// SIMATIC S7-200 SMART project (STEP 7-Micro/WIN SMART), CPU ST40

SYMBOL_TABLE 系统符号
Clock_1s         SM0.5    // 针对 1 s 的周期时间，时钟脉冲接通 0.5 s，断开 0.5 s.
END_SYMBOL_TABLE

ORGANIZATION_BLOCK MAIN:OB1
TITLE=程序注释
BEGIN
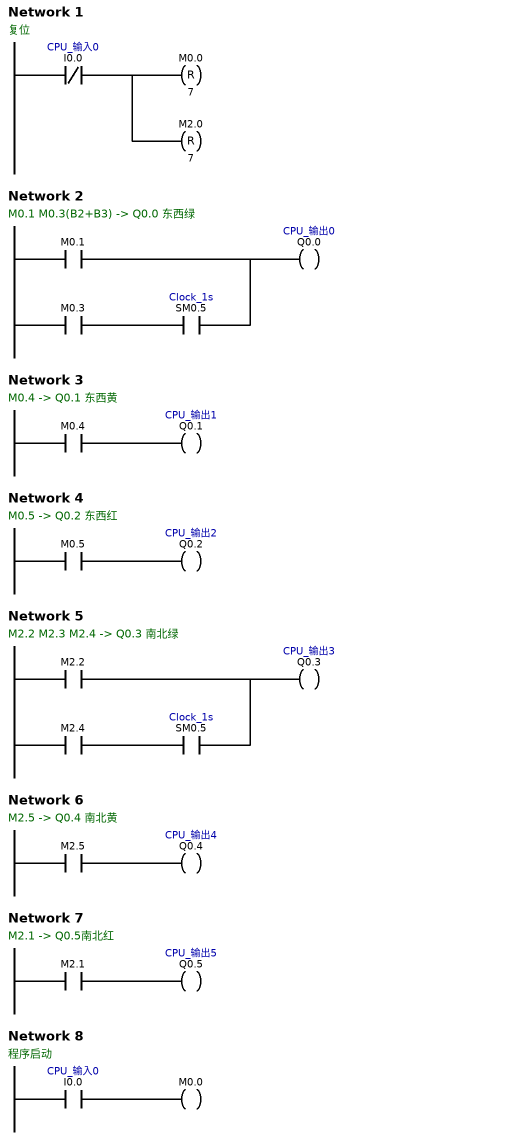
Network 1
// 复位
LDN    CPU_输入0:I0.0
R      M0.0, 7
R      M2.0, 7
Network 2
// M0.1 M0.3(B2+B3) -> Q0.0 东西绿
LD     M0.1
LD     M0.3
A      Clock_1s:SM0.5
OLD
=      CPU_输出0:Q0.0
Network 3
// M0.4 -> Q0.1 东西黄
LD     M0.4
=      CPU_输出1:Q0.1
Network 4
// M0.5 -> Q0.2 东西红
LD     M0.5
=      CPU_输出2:Q0.2
Network 5
// M2.2 M2.3 M2.4 -> Q0.3 南北绿
LD     M2.2
LD     M2.4
A      Clock_1s:SM0.5
OLD
=      CPU_输出3:Q0.3
Network 6
// M2.5 -> Q0.4 南北黄
LD     M2.5
=      CPU_输出4:Q0.4
Network 7
// M2.1 -> Q0.5南北红
LD     M2.1
=      CPU_输出5:Q0.5
Network 8
// 程序启动
LD     CPU_输入0:I0.0
=      M0.0
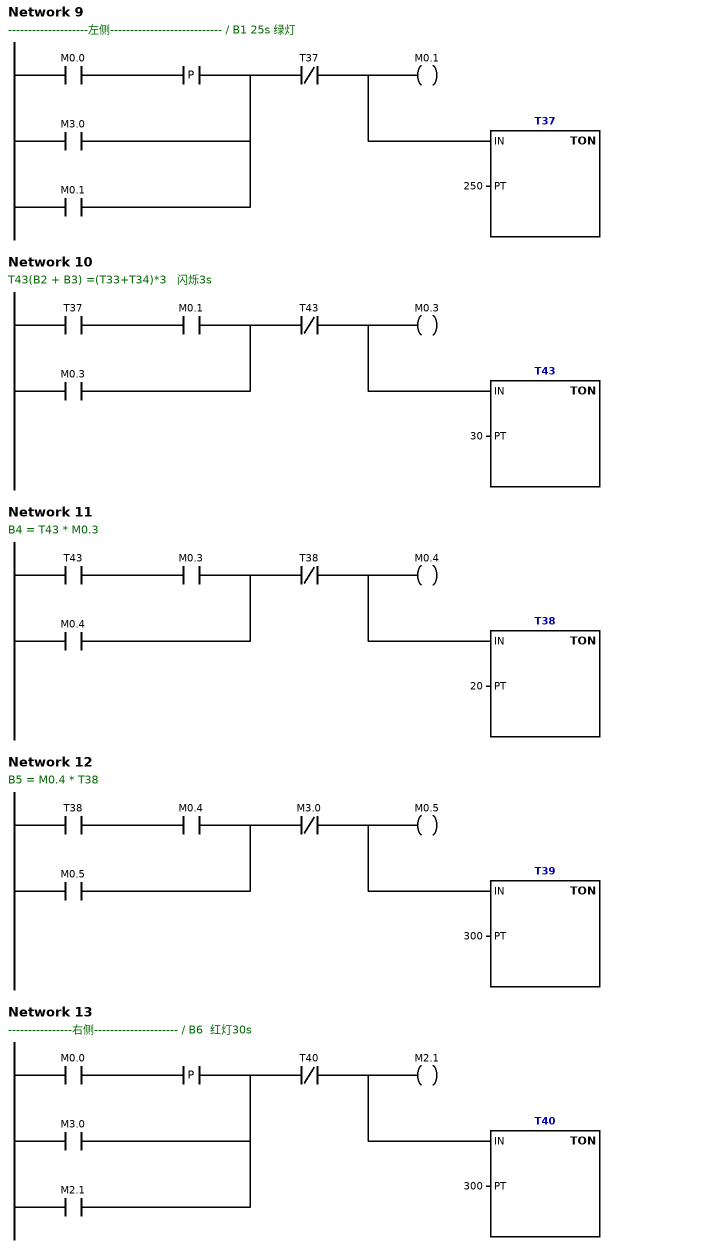
Network 9
// --------------------左侧----------------------------
// B1 25s 绿灯 
LD     M0.0
EU
O      M3.0
O      M0.1
AN     T37
=      M0.1
TON    T37, 250
Network 10
// T43(B2 + B3) =(T33+T34)*3   闪烁3s
LD     T37
A      M0.1
O      M0.3
AN     T43
=      M0.3
TON    T43, 30
Network 11
// B4 = T43 * M0.3
LD     T43
A      M0.3
O      M0.4
AN     T38
=      M0.4
TON    T38, 20
Network 12
// B5 = M0.4 * T38 
LD     T38
A      M0.4
O      M0.5
AN     M3.0
=      M0.5
TON    T39, 300
Network 13
// ----------------右侧---------------------
// B6  红灯30s
LD     M0.0
EU
O      M3.0
O      M2.1
AN     T40
=      M2.1
TON    T40, 300
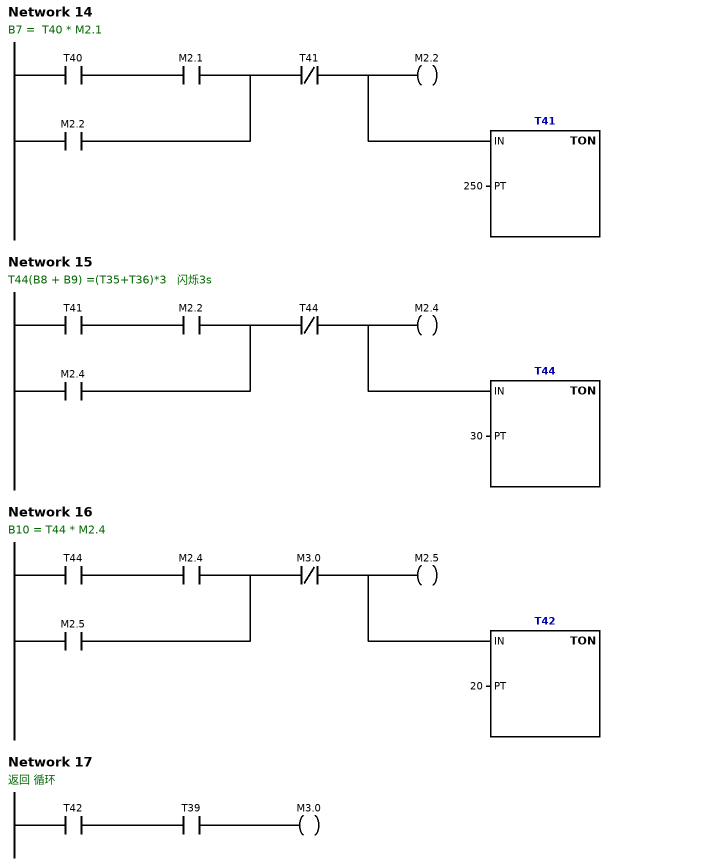
Network 14
// B7 =  T40 * M2.1
LD     T40
A      M2.1
O      M2.2
AN     T41
=      M2.2
TON    T41, 250
Network 15
// T44(B8 + B9) =(T35+T36)*3   闪烁3s
LD     T41
A      M2.2
O      M2.4
AN     T44
=      M2.4
TON    T44, 30
Network 16
// B10 = T44 * M2.4
LD     T44
A      M2.4
O      M2.5
AN     M3.0
=      M2.5
TON    T42, 20
Network 17
// 返回 循环
LD     T42
A      T39
=      M3.0
END_ORGANIZATION_BLOCK
